// TIA Portal V17 export
// export: Created 2024-06-25T12:57:19.2897883Z, ExportSetting WithDefaults, DisplayName Totally Integrated Automation Portal, DisplayVersion V17 Update 6, DisplayName TIA Portal Openness, DisplayVersion V17 Update 6, DisplayName TIA Portal Version Control Interface, DisplayVersion V17, DisplayName STEP 7 Professional, DisplayVersion V17 Update 6, DisplayName STEP 7 Safety, DisplayVersion V17 Update 6, DisplayName WinCC Advanced, DisplayVersion V17 Update 6
VAR_GLOBAL   // PLC tag table "Default tag table"
   F_IN1 AT %I0.0 : Bool;   // SIN / CON PAR
   F_IN2 AT %I0.1 : Bool;   // LLAVIN A MAN/LOC
   F_IN3 AT %I0.2 : Bool;   // LLAVIN A AUTO/REM
   F_IN4 AT %I0.3 : Bool;   // PULSADOR OFF
   F_IN5 AT %I0.4 : Bool;   // PULSADOR MAN
   F_IN6 AT %I0.5 : Bool;   // PULSADOR AUTO
   F_IN7 AT %I0.6 : Bool;   // RES OFF
   F_IN8 AT %I0.7 : Bool;   // RES MAN
   F_IN9 AT %I1.0 : Bool;   // RES AUTO
   F_IN10 AT %I1.1 : Bool;
   F_IN11 AT %I1.2 : Bool;
   F_IN12 AT %I1.3 : Bool;
   F_IN13 AT %I1.4 : Bool;
   F_IN14 AT %I1.5 : Bool;
   F_Q1 AT %Q0.0 : Bool;   // LLAVIN ON
   F_Q2 AT %Q0.1 : Bool;   // LLAVIN AUTO
   F_Q3 AT %Q0.2 : Bool;   // PILOTO OFF
   F_Q4 AT %Q0.3 : Bool;   // PILOTO MAN
   QM1 AT %Q0.4 : Bool;   // PILOTO AUTO
   QM2 AT %Q0.5 : Bool;
   "Q0.6" AT %Q0.6 : Bool;
   "Q0.7" AT %Q0.7 : Bool;
   "Q1.0" AT %Q1.0 : Bool;
   "Q1.1" AT %Q1.1 : Bool;
   "PULSADOR OFF" AT %M0.0 : Bool;
   "PULSADOR AUTO" AT %M0.2 : Bool;
   Tag_1 AT %M200.0 : Bool;
   Tag_2 AT %M200.1 : Bool;
   Tag_3 AT %M200.3 : Bool;
   Tag_4 AT %M200.2 : Bool;
   Tag_5 AT %M200.4 : Bool;
   Tag_6 AT %M200.5 : Bool;
END_VAR
